PROGRAM Comp02_Main

END_PROGRAM

(* stored: Version 1.1.0.1, ProductVersion 3.1.4022.11
   POU Comp02_Main: Id {d7803cdf-0186-480a-b27a-f806155f5a0e}, SpecialFunc None *)
